// TIA Portal V17 program export: 1 tag tables, 0 data types, 1 data blocks, 2 code blocks (in call order from the OBs), 0 instance data blocks

VAR_GLOBAL   // PLC tag table "Default tag table"
END_VAR

DATA_BLOCK "DATOS"   // DB1
{ S7_Optimized_Access := 'TRUE' }
VERSION : 0.1
// stored: AutoNumber true, IsOnlyStoredInLoadMemory false, IsRetainMemResEnabled false, IsWriteProtectedInAS false, MemoryReserve 100
   VAR
      ARRANQUE : Bool;
      PARO : Bool;
      MOTOR : Bool;
      RELE : Bool;
   END_VAR
BEGIN
END_DATA_BLOCK

ORGANIZATION_BLOCK "Main"   // OB1, LAD, ProgramCycle
TITLE = "Main Program Sweep (Cycle)"
{ S7_Optimized_Access := 'TRUE' }
VERSION : 0.1
// stored: AutoNumber true, IsIECCheckEnabled false, SetENOAutomatically false
   VAR_INPUT
      Initial_Call : Bool;   // Initial call of this OB
      Remanence : Bool;   // =True, if remanent data are available
   END_VAR
BEGIN
END_ORGANIZATION_BLOCK

FUNCTION "ARRANQUE DE MOTOR" : Void   // FC1, LAD
{ S7_Optimized_Access := 'TRUE' }
VERSION : 0.1
// stored: AutoNumber true, IsIECCheckEnabled false, SetENOAutomatically false, UDAEnableTagReadback false
BEGIN

REGION Network 1
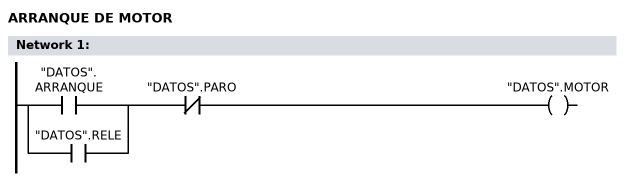
   RUNG wire#powerrail
      Contact( "DATOS".ARRANQUE )
      wire#w1
      I_Contact( "DATOS".PARO )
      Coil( "DATOS".MOTOR )
   END_RUNG
   RUNG wire#powerrail
      Contact( "DATOS".RELE )
   END_RUNG wire#w1
   // the same network as SCL:
   "DATOS".MOTOR := ("DATOS".ARRANQUE OR "DATOS".RELE) AND NOT "DATOS".PARO;
END_REGION
END_FUNCTION
